RoboDK station: P2 - Robot Cell.rdk

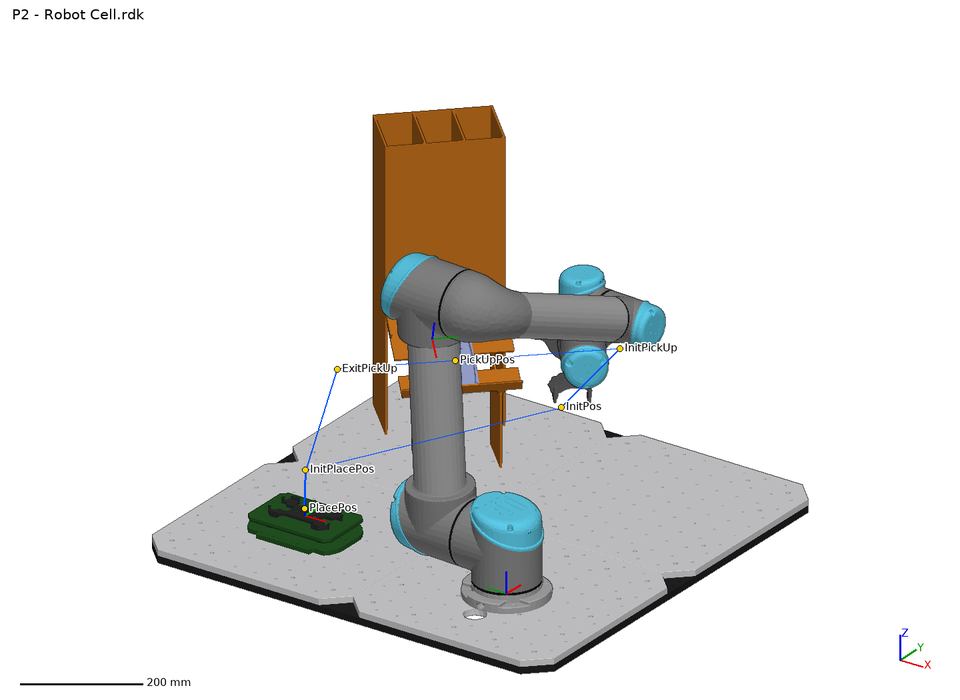
[picture v0: the station drawn from its stored meshes, robots at their saved joint values, targets as dots, program paths as lines]
Station P2 - Robot Cell (saved by RoboDK 5.5.3). Poses are relative to the parent item; angles as X-Y-Z fixed-axis rotations.
  - frame UR5 Base at (0, 0, 0) mm, rotated rx 0 ry 0 rz 90 deg
    - robot UR5: 6 axes
        modified DH rows (alpha deg, a mm, theta deg, d mm): 0, 0, 0, 89.2; 90, 0, 180, 0; 0, 425, 0, 0; 0, 392, 0, 109.3; -90, 0, 0, 94.75; 90, 0, 0, 82.5
        joint limits [-360, -360, -360, -360, -360, -360] to [360, 360, 360, 360, 360, 360]; home [0, -90, -90, 0, 90, 0]; saved at [176.667, -93.648, -243.937, -24.302, 45.969, -83.182]
      - tool GripperAssembled v3, TCP at (120, 0, 0) mm, size 170 x 43.3 x 192 mm, geometry from GripperAssembled v3.step
    - target InitPos (joint target) at (371.96, 152.42, 146.37) mm, rotated rx 120.36 ry 82.55 rz 160.5 deg; joints [177.26, -94.809, -243.076, -16.975, 47.02, -87.07] of UR5
  - object TableTopAssembled at (0, 0, 0) mm, size 800 x 24 x 800 mm, geometry from TableTopAssembled.step
  - frame Pickup Cover at (-414, 381, 194) mm, rotated rx 0.08 ry 24.87 rz -45.72 deg
    - target InitPickUp (joint target) at (56.91, 300, 9.14) mm, rotated rx -5.23 ry 87.74 rz 174.56 deg; joints [175.292, -83.39, 112.154, -66.638, 47.951, -62.679] of UR5
    - target PickUpPos (joint target) at (55.72, 29.25, 8) mm, rotated rx -6.11 ry 87.74 rz 173.65 deg; joints [-152.072, -93.744, 121.513, -55.836, 75.681, -82.701] of UR5
    - target ExitPickUp (joint target) at (54.87, -165.84, 7.18) mm, rotated rx -6.11 ry 87.74 rz 173.65 deg; joints [-123.057, -86.728, 114.595, -55.586, 101.445, -96.165] of UR5
    - object BundCover v1 at (0, 0, 0) mm, size 60 x 114 x 13 mm, geometry from BundCover v1.step
  - frame Place Position at (-400, 0, 30) mm
    - target InitPlacePos (joint target) at (1.28, -1.27, 83.08) mm, rotated rx -7.87 ry 87.97 rz 171.81 deg; joints [-110.073, -97.638, 125.904, -30.406, 70.258, -89.555] of UR5
    - target PlacePos (joint target) at (-1.21, -0.91, 12.3) mm, rotated rx -7.87 ry 87.97 rz 171.81 deg; joints [250.027, -90.24, -228.175, -43.723, 70.359, -89.559] of UR5
    - object PhoneHolder at (0, 0, -30) mm, size 180 x 130 x 46.5 mm, geometry from PhoneHolder.step
  - object BottomCoverDispenser at (-275, 455, 30) mm, rotated rx 0 ry 0 rz 45 deg, size 198 x 282.2 x 529.5 mm, geometry from BottomCoverDispenser.step
  - program Pick&Place (13 instructions, listed below)
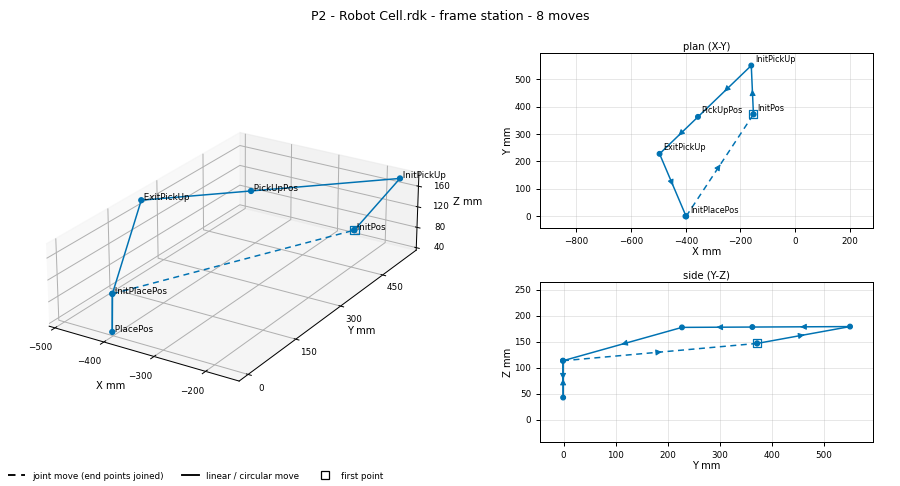
[picture p0: tool path of P2 - Robot Cell.rdk in frame station, 8 of 8 moves have a stored position in this frame; points joined in program order, loops and branches not executed]

--- program Pick&Place (robot UR5) ---
  Set Ref.: Pickup Cover
  Set Tool: GripperAssembled v3
  Replace BundCover v1
  MoveJ (InitPos)
  MoveL (InitPickUp)
  MoveL (PickUpPos)
  Attach to GripperAssembled v3
  MoveL (ExitPickUp)
  MoveL (InitPlacePos)
  MoveL (PlacePos)
  Detach from GripperAssembled v3
  MoveL (InitPlacePos)
  MoveJ (InitPos)
